TYPE DUT_HMI_01_MANUALS :
STRUCT
	PS : ARRAY[0..CNC.NUM_MAX_MANUALS_01-1] OF BOOL;
	LS : ARRAY[0..CNC.NUM_MAX_MANUALS_01-1] OF BOOL;
END_STRUCT
END_TYPE

(* stored: Version 1.1.0.1, ProductVersion 3.1.4024.13
   DUT DUT_HMI_01_MANUALS: Id {e63c6871-a85e-4f24-a8aa-3f0cb3117502} *)
